(************************************************************************************)
(*								Beckhoff Automation Poland							*)
(* 									F_BCDToDec v1.0									*)
(* 										26.06.2014									*)
(*					Funkcja konwertujaca BYTE (kod BCD) na BYTE (DEC)				*)
(*__________________________________________________________________________________*)
FUNCTION F_BCDToDec: BYTE
VAR_INPUT
	BIn:BYTE;
END_VAR

CASE ROL(BIn AND 16#F0,4) OF
0:	F_BCDToDec := 00;
1:	F_BCDToDec := 10;
2:	F_BCDToDec := 20;
3:	F_BCDToDec := 30;
4:	F_BCDToDec := 40;
5:	F_BCDToDec := 50;
6:	F_BCDToDec := 60;
7:	F_BCDToDec := 70;
8:	F_BCDToDec := 80;
9:	F_BCDToDec := 90;
ELSE
	;
END_CASE

CASE BIn AND 16#F OF
0..9:	F_BCDToDec := F_BCDToDec + (BIn AND 16#F);
ELSE
	;
END_CASE

END_FUNCTION

(* stored: Version 1.1.0.1, ProductVersion 3.1.4026.13, FileIdentifier d2547641f7d94ce354245263c474f7010d6eb956, FileSignature 800c887b58289993fc87ccac59f1051cf36f4b65894f7cbbf5c9a3a7f968a2abd069b26a40a831b4f0a6817453e01d2e06e513051cbc5f774d88c705eea6e1318f71dda06ba7b568541eb970eb45578a37628426cc456282386a6c3ecdc8f241b9d3841eb1c7ada14dbd7c91f230513cd2e51841fe387865a9217f8e748f86a12f731c477bf7813916ab685c8ec37cd69b8e293f88c066591ef5a21e662901ea2c335f5f9868c874f0c68eb4ca3007eb4730eae45d267f06752e4ad26addcbcc6b3623bbc7c045c0d47518640cf7034cc86f70cde2077e212518548ff8b19676cb7f22d6c1d0f1665b0da98e70e9e69104fde99eb71df003acafaf8d1eabe3bd
   POU F_BCDToDec: Id {8ba2a411-6671-4d19-aa23-08ab68f2c827}, SpecialFunc None *)
